// TIA Portal V17 export
// export: Created 2023-03-22T09:20:33.7548981Z, ExportSetting WithDefaults, DisplayName Totally Integrated Automation Portal, DisplayVersion V17 Update 4, DisplayName TIA Portal Openness, DisplayVersion V17 Update 4, DisplayName TIA Portal Version Control Interface, DisplayVersion V17, DisplayName STEP 7 Professional, DisplayVersion V17 Update 4, DisplayName STEP 7 Safety, DisplayVersion V17, DisplayName WinCC Professional, DisplayVersion V17 Update 4
FUNCTION "SS Alarms" : Void   // FC102, LAD
{ S7_Optimized_Access := 'TRUE' }
VERSION : 0.1
// stored: AutoNumber false, IsIECCheckEnabled false, SetENOAutomatically false, UDAEnableTagReadback false
BEGIN

REGION Network 1: Alarm Status On/Off
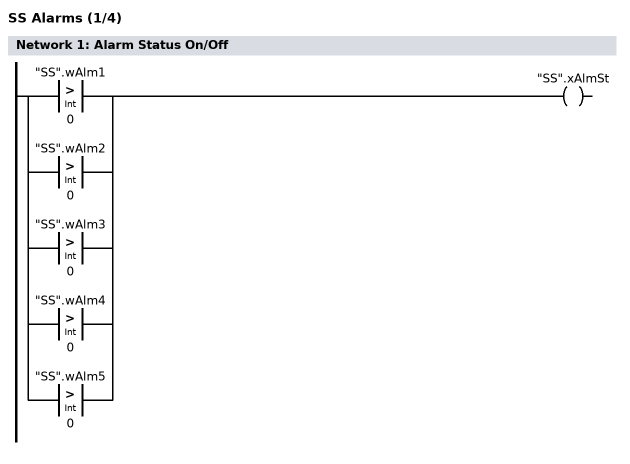
   RUNG wire#powerrail
      { S7_Templates := "SrcType := Int" } GT_Contact(in1 := "SS".wAlm1, in2 := 0)
      wire#w1
      Coil( "SS".xAlmSt )
   END_RUNG
   RUNG wire#powerrail
      { S7_Templates := "SrcType := Int" } GT_Contact(in1 := "SS".wAlm2, in2 := 0)
   END_RUNG wire#w1
   RUNG wire#powerrail
      { S7_Templates := "SrcType := Int" } GT_Contact(in1 := "SS".wAlm3, in2 := 0)
   END_RUNG wire#w1
   RUNG wire#powerrail
      { S7_Templates := "SrcType := Int" } GT_Contact(in1 := "SS".wAlm4, in2 := 0)
   END_RUNG wire#w1
   RUNG wire#powerrail
      { S7_Templates := "SrcType := Int" } GT_Contact(in1 := "SS".wAlm5, in2 := 0)
   END_RUNG wire#w1
   // the same network as SCL:
   "SS".xAlmSt := ("SS".wAlm1 > 0) OR ("SS".wAlm2 > 0) OR ("SS".wAlm3 > 0) OR ("SS".wAlm4 > 0) OR ("SS".wAlm5 > 0);
END_REGION

REGION Network 2: Alarm Word 1
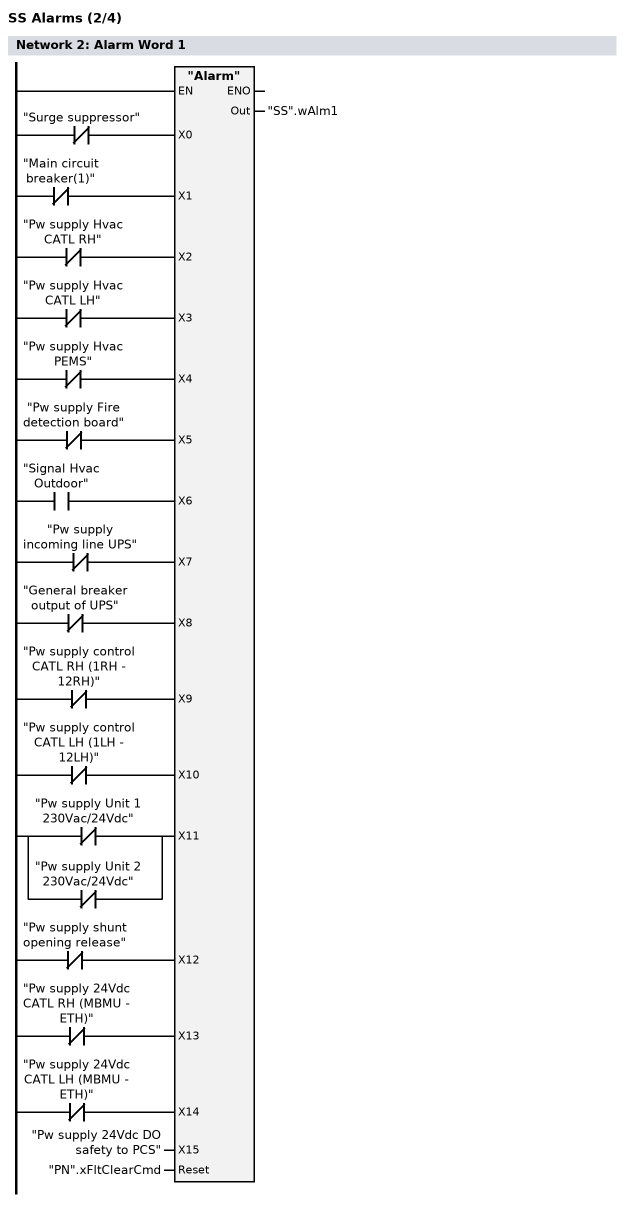
   RUNG wire#powerrail
      "Alarm"(X0 := wire#w1, X1 := wire#w2, X2 := wire#w3, X3 := wire#w4, X4 := wire#w5, X5 := wire#w6, X6 := wire#w7, X7 := wire#w8, X8 := wire#w9, X9 := wire#w10, X10 := wire#w11, X11 := wire#w12, X12 := wire#w13, X13 := wire#w14, X14 := wire#w15, X15 := "Pw supply 24Vdc DO safety to PCS", Reset := "PN".xFltClearCmd, Out => "SS".wAlm1)
   END_RUNG
   RUNG wire#powerrail
      I_Contact( "Surge suppressor" )
   END_RUNG wire#w1
   RUNG wire#powerrail
      I_Contact( "Main circuit breaker(1)" )
   END_RUNG wire#w2
   RUNG wire#powerrail
      I_Contact( "Pw supply Hvac CATL RH" )
   END_RUNG wire#w3
   RUNG wire#powerrail
      I_Contact( "Pw supply Hvac CATL LH" )
   END_RUNG wire#w4
   RUNG wire#powerrail
      I_Contact( "Pw supply Hvac PEMS" )
   END_RUNG wire#w5
   RUNG wire#powerrail
      I_Contact( "Pw supply Fire detection board" )
   END_RUNG wire#w6
   RUNG wire#powerrail
      Contact( "Signal Hvac Outdoor" )
   END_RUNG wire#w7
   RUNG wire#powerrail
      I_Contact( "Pw supply incoming line UPS" )
   END_RUNG wire#w8
   RUNG wire#powerrail
      I_Contact( "General breaker output of UPS" )
   END_RUNG wire#w9
   RUNG wire#powerrail
      I_Contact( "Pw supply control CATL RH (1RH - 12RH)" )
   END_RUNG wire#w10
   RUNG wire#powerrail
      I_Contact( "Pw supply control CATL LH (1LH - 12LH)" )
   END_RUNG wire#w11
   RUNG wire#powerrail
      I_Contact( "Pw supply Unit 1 230Vac/24Vdc" )
   END_RUNG wire#w12
   RUNG wire#powerrail
      I_Contact( "Pw supply Unit 2 230Vac/24Vdc" )
   END_RUNG wire#w12
   RUNG wire#powerrail
      I_Contact( "Pw supply shunt opening release" )
   END_RUNG wire#w13
   RUNG wire#powerrail
      I_Contact( "Pw supply 24Vdc CATL RH (MBMU - ETH)" )
   END_RUNG wire#w14
   RUNG wire#powerrail
      I_Contact( "Pw supply 24Vdc CATL LH (MBMU - ETH)" )
   END_RUNG wire#w15
   // the same network as SCL:
   "Alarm"(X0 := NOT "Surge suppressor",
           X1 := NOT "Main circuit breaker(1)",
           X2 := NOT "Pw supply Hvac CATL RH",
           X3 := NOT "Pw supply Hvac CATL LH",
           X4 := NOT "Pw supply Hvac PEMS",
           X5 := NOT "Pw supply Fire detection board",
           X6 := "Signal Hvac Outdoor",
           X7 := NOT "Pw supply incoming line UPS",
           X8 := NOT "General breaker output of UPS",
           X9 := NOT "Pw supply control CATL RH (1RH - 12RH)",
           X10 := NOT "Pw supply control CATL LH (1LH - 12LH)",
           X11 := NOT "Pw supply Unit 1 230Vac/24Vdc" OR NOT "Pw supply Unit 2 230Vac/24Vdc",
           X12 := NOT "Pw supply shunt opening release",
           X13 := NOT "Pw supply 24Vdc CATL RH (MBMU - ETH)",
           X14 := NOT "Pw supply 24Vdc CATL LH (MBMU - ETH)",
           X15 := "Pw supply 24Vdc DO safety to PCS",
           Reset := "PN".xFltClearCmd,
           Out => "SS".wAlm1);
END_REGION

REGION Network 3: Alarm Word 2
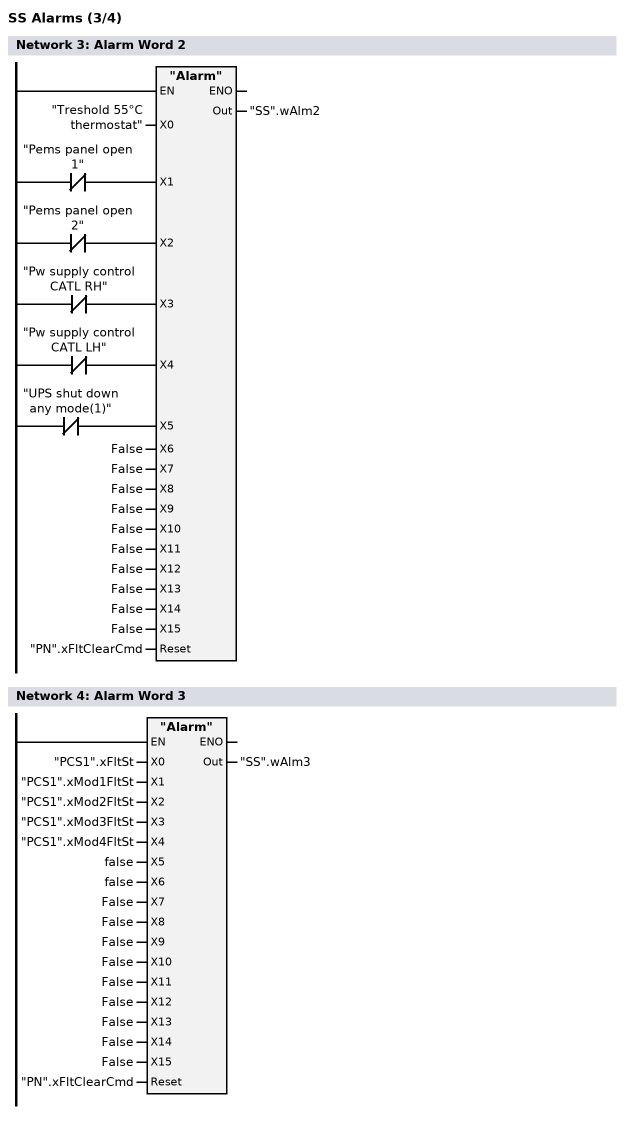
   RUNG wire#powerrail
      "Alarm"(X1 := wire#w1, X2 := wire#w2, X3 := wire#w3, X4 := wire#w4, X5 := wire#w5, X0 := "Treshold 55°C thermostat", X6 := False, X7 := False, X8 := False, X9 := False, X10 := False, X11 := False, X12 := False, X13 := False, X14 := False, X15 := False, Reset := "PN".xFltClearCmd, Out => "SS".wAlm2)
   END_RUNG
   RUNG wire#powerrail
      I_Contact( "Pems panel open 1" )
   END_RUNG wire#w1
   RUNG wire#powerrail
      I_Contact( "Pems panel open 2" )
   END_RUNG wire#w2
   RUNG wire#powerrail
      I_Contact( "Pw supply control CATL RH" )
   END_RUNG wire#w3
   RUNG wire#powerrail
      I_Contact( "Pw supply control CATL LH" )
   END_RUNG wire#w4
   RUNG wire#powerrail
      I_Contact( "UPS shut down any mode(1)" )
   END_RUNG wire#w5
   // the same network as SCL:
   "Alarm"(X0 := "Treshold 55°C thermostat",
           X1 := NOT "Pems panel open 1",
           X2 := NOT "Pems panel open 2",
           X3 := NOT "Pw supply control CATL RH",
           X4 := NOT "Pw supply control CATL LH",
           X5 := NOT "UPS shut down any mode(1)",
           X6 := False,
           X7 := False,
           X8 := False,
           X9 := False,
           X10 := False,
           X11 := False,
           X12 := False,
           X13 := False,
           X14 := False,
           X15 := False,
           Reset := "PN".xFltClearCmd,
           Out => "SS".wAlm2);
END_REGION

REGION Network 4: Alarm Word 3
   RUNG wire#powerrail
      "Alarm"(X0 := "PCS1".xFltSt, X1 := "PCS1".xMod1FltSt, X2 := "PCS1".xMod2FltSt, X3 := "PCS1".xMod3FltSt, X4 := "PCS1".xMod4FltSt, X5 := false, X6 := false, X7 := False, X8 := False, X9 := False, X10 := False, X11 := False, X12 := False, X13 := False, X14 := False, X15 := False, Reset := "PN".xFltClearCmd, Out => "SS".wAlm3)
   END_RUNG
   // the same network as SCL:
   "Alarm"(X0 := "PCS1".xFltSt,
           X1 := "PCS1".xMod1FltSt,
           X2 := "PCS1".xMod2FltSt,
           X3 := "PCS1".xMod3FltSt,
           X4 := "PCS1".xMod4FltSt,
           X5 := false,
           X6 := false,
           X7 := False,
           X8 := False,
           X9 := False,
           X10 := False,
           X11 := False,
           X12 := False,
           X13 := False,
           X14 := False,
           X15 := False,
           Reset := "PN".xFltClearCmd,
           Out => "SS".wAlm3);
END_REGION

REGION Network 5: Alarm Word 4
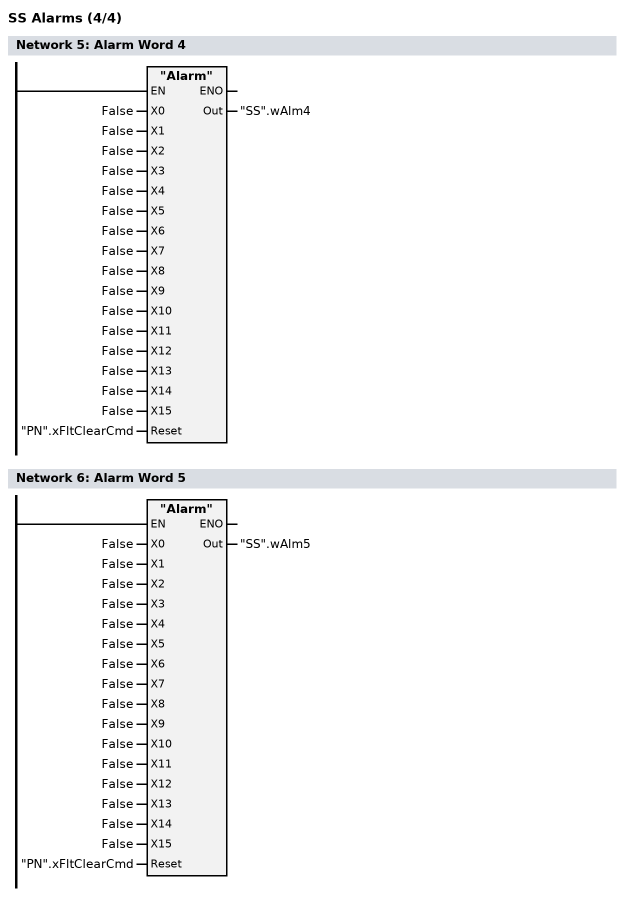
   RUNG wire#powerrail
      "Alarm"(X0 := False, X1 := False, X2 := False, X3 := False, X4 := False, X5 := False, X6 := False, X7 := False, X8 := False, X9 := False, X10 := False, X11 := False, X12 := False, X13 := False, X14 := False, X15 := False, Reset := "PN".xFltClearCmd, Out => "SS".wAlm4)
   END_RUNG
   // the same network as SCL:
   "Alarm"(X0 := False,
           X1 := False,
           X2 := False,
           X3 := False,
           X4 := False,
           X5 := False,
           X6 := False,
           X7 := False,
           X8 := False,
           X9 := False,
           X10 := False,
           X11 := False,
           X12 := False,
           X13 := False,
           X14 := False,
           X15 := False,
           Reset := "PN".xFltClearCmd,
           Out => "SS".wAlm4);
END_REGION

REGION Network 6: Alarm Word 5
   RUNG wire#powerrail
      "Alarm"(X0 := False, X1 := False, X2 := False, X3 := False, X4 := False, X5 := False, X6 := False, X7 := False, X8 := False, X9 := False, X10 := False, X11 := False, X12 := False, X13 := False, X14 := False, X15 := False, Reset := "PN".xFltClearCmd, Out => "SS".wAlm5)
   END_RUNG
   // the same network as SCL:
   "Alarm"(X0 := False,
           X1 := False,
           X2 := False,
           X3 := False,
           X4 := False,
           X5 := False,
           X6 := False,
           X7 := False,
           X8 := False,
           X9 := False,
           X10 := False,
           X11 := False,
           X12 := False,
           X13 := False,
           X14 := False,
           X15 := False,
           Reset := "PN".xFltClearCmd,
           Out => "SS".wAlm5);
END_REGION
END_FUNCTION
